PROGRAM MAIN
VAR
	//SThisIsOurFirstInstanceOfAStructure : ST_Event;
	bBoolean : BOOL := False;
	eEventType1 : E_EventType := E_EventType.Alarm;
	eEventSeverity1 : TcEventSeverity := TcEventSeverity.Error;
	nEventIdentity1 : UDINT := 42;
	sEventText1 : STRING(255) := 'En détente';
	CsvPersistentEventStorage : FB_CsvPersistentEventStorage;
	EventLogger : EventLogger(CsvPersistentEventStorage);
END_VAR

(*
IF NOT bBoolean THEN 
	UpdateEventTimestampWithSystemTime(stEvent := SThisIsOurFirstInstanceOfAStructure);
	bBoolean := TRUE;
END_IF
*)
IF bBoolean THEN 
	EventLogger.AddEvent(eEventType1,  eEventSeverity1, nEventIdentity1, sEventText1);
	bBoolean := FALSE;
	//here we will add the event
END_IF

CsvPersistentEventStorage();

// a comment

END_PROGRAM

(* stored: Version 1.1.0.1, ProductVersion 3.1.4024.12
   POU MAIN: Id {44073901-dcdc-48ee-ba3b-ef20bef62b8d}, SpecialFunc None *)
